(* CoDeSys 2.3.9.28 project: AULA05_EX02.pro *)
(* Libraries: Standard.lib 27.1.09 11:27:38, Util.lib 27.1.09 11:27:38, IecSfc.lib*24.11.08 08:07:15, SysLibTime.lib*27.1.09 11:27:38, SysTaskInfo.lib 24.11.08 08:07:15, SYSLIBCALLBACK.LIB 27.1.09 11:27:38 *)

(* PLC configuration (modules and I/O channels)
Hexswitch AT %IB0 [HexSwitch] rotary switch 0 = STOP, 1-15 = RUN
IOModules [CPX_MASTER] node 0, in %IB4 out %QB0
  8DI/8DO [CPX-8DI_8DO_Multi_I_O_module_1] node 0, in %IB4 out %QB0 {StringParam = 4,8,1,8,1; ByteParam = 7; ByteParam = 81; ByteParam = 0; ByteParam = 0; ByteParam = 0; ByteParam = 0; ByteParam = 0; IdleStateParam = 0; IdleModeParam = 255; IdleStateParam = 0; IdleModeParam = 255; IdleStateParam = 0; IdleModeParam = 255; IdleStateParam = 0; IdleModeParam = 255}
    AT %IB4 [ByteInput] -
    AT %QB0 [ByteOutput] -
  8DI/8DO [CPX-8DI_8DO_Multi_I_O_module_1] node 1, in %IB8 out %QB4 {StringParam = 4,8,1,8,1; ByteParam = 7; ByteParam = 81; ByteParam = 0; ByteParam = 0; ByteParam = 0; ByteParam = 0; ByteParam = 0; IdleStateParam = 0; IdleModeParam = 255; IdleStateParam = 0; IdleModeParam = 255; IdleStateParam = 0; IdleModeParam = 255; IdleStateParam = 0; IdleModeParam = 255}
    AT %IB8 [ByteInput] -
    AT %QB4 [ByteOutput] -
*)

(* Global variable list: Global_Variables *)
VAR_GLOBAL

	START AT %IX2.0 : BOOL;
	STOP AT %IX2.1 : BOOL;
	S1 AT %IX2.2 : BOOL;
	S2 AT %IX2.3 : BOOL;
	S3 AT %IX2.4 : BOOL;
	S4 AT %IX2.5 : BOOL;
	S5 AT %IX2.6 : BOOL;

	LAMP AT %QX0.0 : BOOL;
	M1 AT %QX0.1 : BOOL;
	C1 AT %QX0.2 : BOOL;
	C2 AT %QX0.3 : BOOL;

END_VAR

(* POU PLC_PRG, LD *)
PROGRAM PLC_PRG
VAR
END_VAR
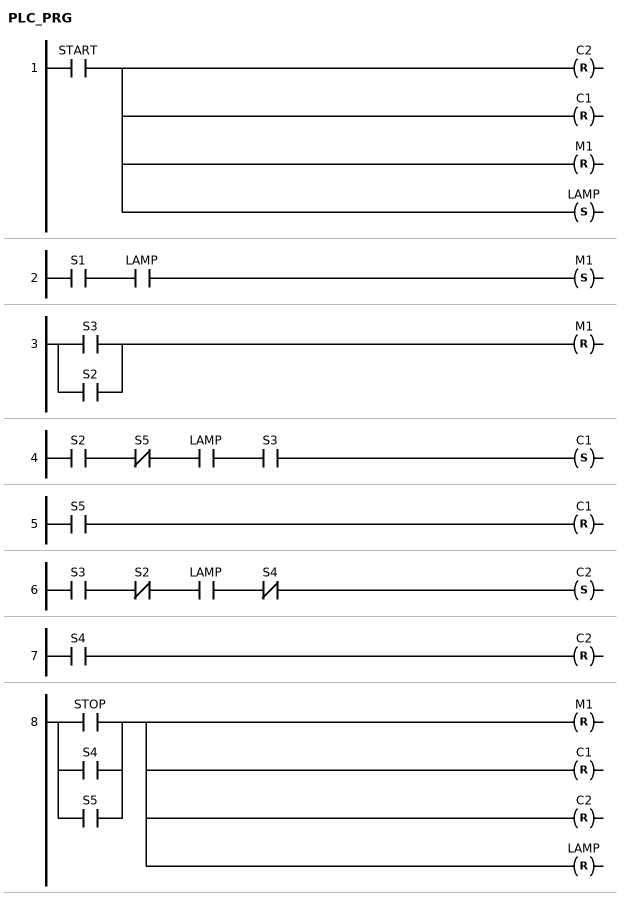
_LD_ (* Ladder Diagram *)
NETWORK 1
	[START] --- (R C2) (R C1) (R M1) (S LAMP)
NETWORK 2
	[S1] - [LAMP] --- (S M1)
NETWORK 3
	{ [S3] | [S2] } --- (R M1)
NETWORK 4
	[S2] - [/S5] - [LAMP] - [S3] --- (S C1)
NETWORK 5
	[S5] --- (R C1)
NETWORK 6
	[S3] - [/S2] - [LAMP] - [/S4] --- (S C2)
NETWORK 7
	[S4] --- (R C2)
NETWORK 8
	{ [STOP] | [S4] | [S5] } --- (R M1) (R C1) (R C2) (R LAMP)
_END_LD_
(* the same logic as Structured Text *)
(* Network 1 *)
IF START THEN C2 := FALSE; C1 := FALSE; M1 := FALSE; LAMP := TRUE; END_IF;
(* Network 2 *)
IF S1 AND LAMP THEN M1 := TRUE; END_IF;
(* Network 3 *)
IF S3 OR S2 THEN M1 := FALSE; END_IF;
(* Network 4 *)
IF S2 AND NOT S5 AND LAMP AND S3 THEN C1 := TRUE; END_IF;
(* Network 5 *)
IF S5 THEN C1 := FALSE; END_IF;
(* Network 6 *)
IF S3 AND NOT S2 AND LAMP AND NOT S4 THEN C2 := TRUE; END_IF;
(* Network 7 *)
IF S4 THEN C2 := FALSE; END_IF;
(* Network 8 *)
IF STOP OR S4 OR S5 THEN M1 := FALSE; C1 := FALSE; C2 := FALSE; LAMP := FALSE; END_IF;
END_PROGRAM
